GLOBALCONSTANTS AID_IB (* Input boolean object attribute ids *)
  (* Standard: 61499-1; Description: Copyright (c) 2023 HR Agrartechnik GmbH This program and the accompanying materials are made available under the terms of the Eclipse Public License 2.0 which is available at https://www.eclipse.org/legal/epl-2.0/ SPDX-License-Identifier: EPL-2.0 *)
  (* Version 1.0, 2026-06-20, Franz Höpfinger, HR Agrartechnik GmbH *)
  PACKAGE isobus::UT::Q::const::AID;
  VAR_GLOBAL CONSTANT
    BACKGROUND_COLOUR : USINT := USINT#1; (* 1: AID_IB_BACKGROUND_COLOUR - Background colour index. *)
    WIDTH : USINT := USINT#2; (* 2: AID_IB_WIDTH - Width in pixels. *)
    FG_COLOUR : USINT := USINT#3; (* 3: AID_IB_FG_COLOUR - Object ID of a Font Attributes object to use for font colour. *)
    VARIABLE_REF : USINT := USINT#4; (* 4: AID_IB_VARIABLE_REF - Object ID of a Number Variable object. If NULL, value is stored *)
    VALUE : USINT := USINT#5; (* 5: AID_IB_VALUE - Value of the input field: 0 for FALSE, >0 for TRUE. *)
    ENABLED : USINT := USINT#6; (* 6: AID_IB_ENABLED - 0 = Disabled, 1 = Enabled. *)
  END_VAR
END_GLOBALCONSTANTS
